FUNCTION_BLOCK JobMgr
VAR_INPUT
	Cmd:	JobCmd_typ;
	rXTS:	REFERENCE TO XTSMainControl_typ;
	rRecoveryZone: REFERENCE TO Zone;
END_VAR
VAR_OUTPUT
	Sts:		JobSts_typ;
END_VAR
VAR
	State:		JobState_enum;
	Orient:		JobStn_typ;
	BallSeat:	JobStn_typ;
	Print:		JobStn_typ;
	Vision:		JobStn_typ;
	Kickout:	JobStn_typ;
	TrayLoad:	JobStn_typ;
	System:		JobStn_typ;

	StnCmdRun:	BOOL;
	StnStsAllNotRunning: BOOL;
	Payload	: Payload_typ;

	_State:		JobState_enum;
	i: INT;
END_VAR

CASE State OF
	Job_Disabled:
		IF _State <> Job_Disabled THEN
			;//Clear Job Statuses and Counts
		END_IF

		IF Cmd.Run AND rXTS.Sts.Enabled THEN
			StnCmdRun	:= TRUE;
			State		:= Job_Running;
		END_IF

	Job_Starting:
		;

	Job_Running:
		IF Sts.Done THEN
			StnCmdRun	:= FALSE;
			State		:= Job_Done;
		ELSIF Cmd.Cleanout OR NOT Cmd.Run THEN
			StnCmdRun	:= FALSE;
			State		:= Job_Pausing;
		END_IF

	Job_Pausing:
		IF Cmd.Run THEN
			StnCmdRun	:= TRUE;
			State		:= Job_Running;
		ELSIF Cmd.Cleanout AND StnStsAllNotRunning THEN
			;//MEMSET(rjo
		END_IF

	Job_Paused:
		IF Cmd.Run THEN
			StnCmdRun	:= TRUE;
			State		:= Job_Running;
		ELSIF Cmd.Cleanout THEN
			StnCmdRun	:= FALSE;
			//Sts. 
		END_IF

	Job_Done:
		IF NOT Cmd.Run THEN
			State	:= Job_Disabled;
		END_IF

	Job_Cleanout:
		IF Sts.CleanoutDone AND NOT Cmd.Cleanout THEN
			State	:= Job_Disabled;
		END_IF
END_CASE;

// Stn Commands
Orient.Cmd.Run := BallSeat.Cmd.Run := Print.Cmd.Run := StnCmdRun := Vision.Cmd.Run := Kickout.Cmd.Run := TrayLoad.Cmd.Run := StnCmdRun;

// Stn Specific Commands
FOR i := 0 TO 3 DO
	Orient.Cmd.PlayerNumberCount[i]	:= (Cmd.PlayerNumberCount[0] * 12) + Sts.RejectedPlayerNumberCount[i];
END_FOR
Print.Cmd.NumColor		:= Cmd.NumColor;
Print.Cmd.NumIndex		:= Cmd.NumIndex;
Print.Cmd.IgnoreVision	:= Cmd.IgnoreVision;
Vision.Cmd.IgnoreVision	:= Cmd.IgnoreVision;

// Stn Statuses
StnStsAllNotRunning := NOT (Orient.Sts.Running OR BallSeat.Sts.Running OR Print.Sts.Running OR Vision.Sts.Running OR Kickout.Sts.Running OR TrayLoad.Sts.Running);

// Outputs
Sts.Running						:= State = Job_Running;
Sts.Done						:= State = Job_Done;
Sts.PlayerNumberCount			:= TrayLoad.Sts.PlayerNumberCount;
Sts.PrintedPlayerNumberCount	:= Print.Sts.PlayerNumberCount;
FOR i := 0 TO 3 DO
Sts.RejectedPlayerNumberCount[i]	:= Orient.Sts.RejectedPlayerNumberCount[i] + BallSeat.Sts.RejectedPlayerNumberCount[i] +
									Print.Sts.RejectedPlayerNumberCount[i] + Vision.Sts.RejectedPlayerNumberCount[i] +
									Kickout.Sts.RejectedPlayerNumberCount[i] + Trayload.Sts.RejectedPlayerNumberCount[i] +
									System.Sts.RejectedPlayerNumberCount[i];
END_FOR

// Save Previous Values
_State	:= State;

END_FUNCTION_BLOCK

(* stored: Version 1.1.0.1, ProductVersion 3.1.4024.12
   POU JobMgr: Id {bc0b6362-74f3-0105-0ef2-523b606f0192}, SpecialFunc None *)
